FUNCTION_BLOCK FINAL FB_ServoMove
VAR_INPUT
	ExecuteMove					: BOOL;					
END_VAR
VAR_IN_OUT
	Axis						: AXIS_REF;				
	PosMove						: ST_MovePosition_SP;
	CMD_MovePosAbs				: MC_MOVEABSOLUTE;
	CMD_MovePosMod				: MC_MOVEMODULO;
	CMD_MovePosRel				: MC_MOVERELATIVE;	
END_VAR
VAR
	_accelRate					: LREAL;
	_decelRate					: LREAL;
	_jerkTime					: REAL;
	_jerkValue					: LREAL;
	_posMoveAbsActive			: BOOL;
	_posMoveRelActive			: BOOL;
	_posMoveModActive			: BOOL;
END_VAR

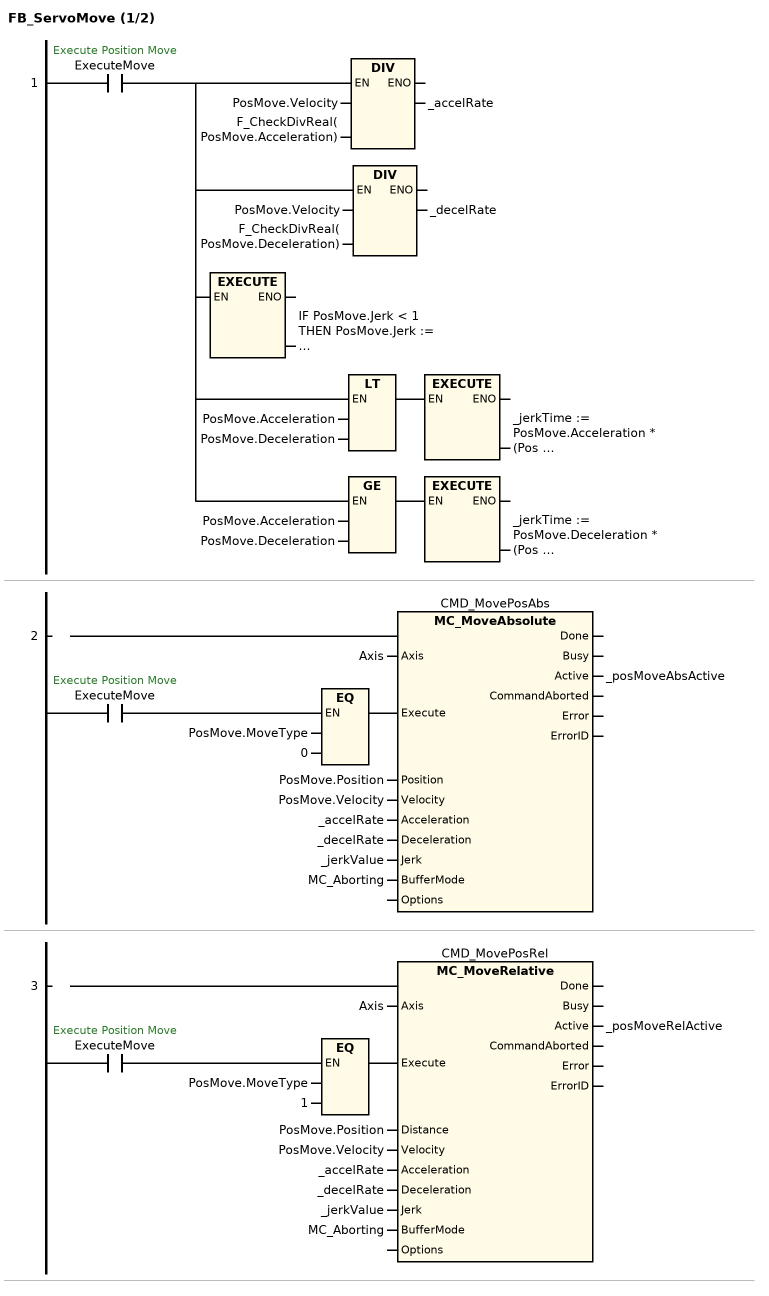
// NETWORK 1
//   ExecuteMove: Execute Position Move
//   PosMove.Velocity: Velocity Value of Move
//   F_CheckDivReal(PosMove.Acceleration): Accleration Value of Move
//   F_CheckDivReal(PosMove.Deceleration): Deceleration Value of Move
//   PosMove.Acceleration: Accleration Value of Move
//   PosMove.Deceleration: Deceleration Value of Move
IF ExecuteMove THEN _accelRate := PosMove.Velocity / (F_CheckDivReal(PosMove.Acceleration)); END_IF
IF ExecuteMove THEN _decelRate := PosMove.Velocity / (F_CheckDivReal(PosMove.Deceleration)); END_IF
IF ExecuteMove THEN
    IF PosMove.Jerk < 1 THEN PosMove.Jerk := 1; END_IF
    IF PosMove.Jerk > 100 THEN PosMove.Jerk := 100; END_IF
END_IF
IF ExecuteMove AND PosMove.Acceleration < PosMove.Deceleration THEN
    _jerkTime := PosMove.Acceleration * (PosMove.Jerk / 100);
    _jerkValue := _accelRate / F_CheckDivReal(_jerkTime);
END_IF
IF ExecuteMove AND PosMove.Acceleration >= PosMove.Deceleration THEN
    _jerkTime := PosMove.Deceleration * (PosMove.Jerk / 100);
    _jerkValue := _decelRate / F_CheckDivReal(_jerkTime);
END_IF

// NETWORK 2
//   ExecuteMove: Execute Position Move
//   PosMove.MoveType: Move Type Configuration of Positional Move
//   PosMove.Position: Position Value to Move to
//   PosMove.Velocity: Velocity Value of Move
CMD_MovePosAbs(
    Axis := Axis,
    Execute := ExecuteMove AND PosMove.MoveType = 0,
    Position := PosMove.Position,
    Velocity := PosMove.Velocity,
    Acceleration := _accelRate,
    Deceleration := _decelRate,
    Jerk := _jerkValue,
    BufferMode := MC_Aborting,
    Active => _posMoveAbsActive); // MC_MoveAbsolute

// NETWORK 3
//   ExecuteMove: Execute Position Move
//   PosMove.MoveType: Move Type Configuration of Positional Move
//   PosMove.Position: Position Value to Move to
//   PosMove.Velocity: Velocity Value of Move
CMD_MovePosRel(
    Axis := Axis,
    Execute := ExecuteMove AND PosMove.MoveType = 1,
    Distance := PosMove.Position,
    Velocity := PosMove.Velocity,
    Acceleration := _accelRate,
    Deceleration := _decelRate,
    Jerk := _jerkValue,
    BufferMode := MC_Aborting,
    Active => _posMoveRelActive); // MC_MoveRelative

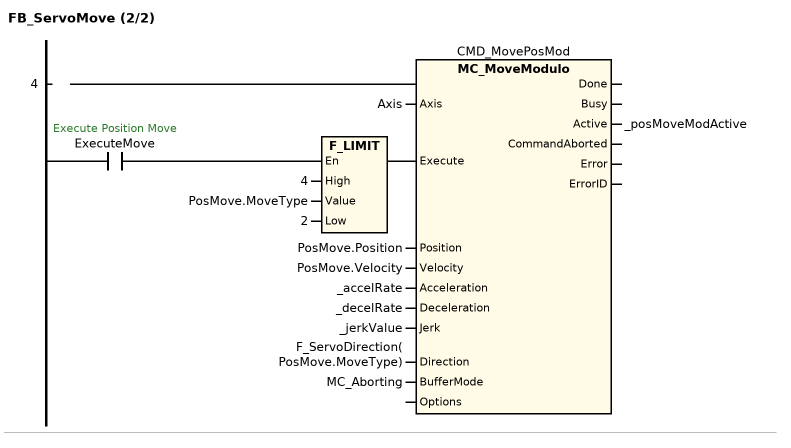
// NETWORK 4
//   ExecuteMove: Execute Position Move
//   PosMove.MoveType: Move Type Configuration of Positional Move
//   PosMove.Position: Position Value to Move to
//   PosMove.Velocity: Velocity Value of Move
CMD_MovePosMod(
    Axis := Axis,
    Execute := F_LIMIT(En := ExecuteMove, High := 4, Value := PosMove.MoveType, Low := 2),
    Position := PosMove.Position,
    Velocity := PosMove.Velocity,
    Acceleration := _accelRate,
    Deceleration := _decelRate,
    Jerk := _jerkValue,
    Direction := F_ServoDirection(PosMove.MoveType),
    BufferMode := MC_Aborting,
    Active => _posMoveModActive); // MC_MoveModulo

END_FUNCTION_BLOCK

(* stored: Version 1.1.0.1, ProductVersion 3.1.4024.3
   POU FB_ServoMove: Id {91ffa93b-025f-4478-8aac-fc1cacc7ffb6}, SpecialFunc None *)
